SUBAPPLICATION Versuch_406 (* Versuch Array Summe *)
  (* Standard: 61499-2; Description: Copyright (c) 2023 Meisterschulen am Ostbahnhof This program and the accompanying materials are made available under the terms of the Eclipse Public License 2.0 which is available at https://www.eclipse.org/legal/epl-2.0/ SPDX-License-Identifier: EPL-2.0 *)
  (* Version 1.0, 2023-10-23, Franz Höpfinger, Meisterschulen am Ostbahnhof, initial API and implementation and/or initial documentation *)
  PACKAGE Versuche;
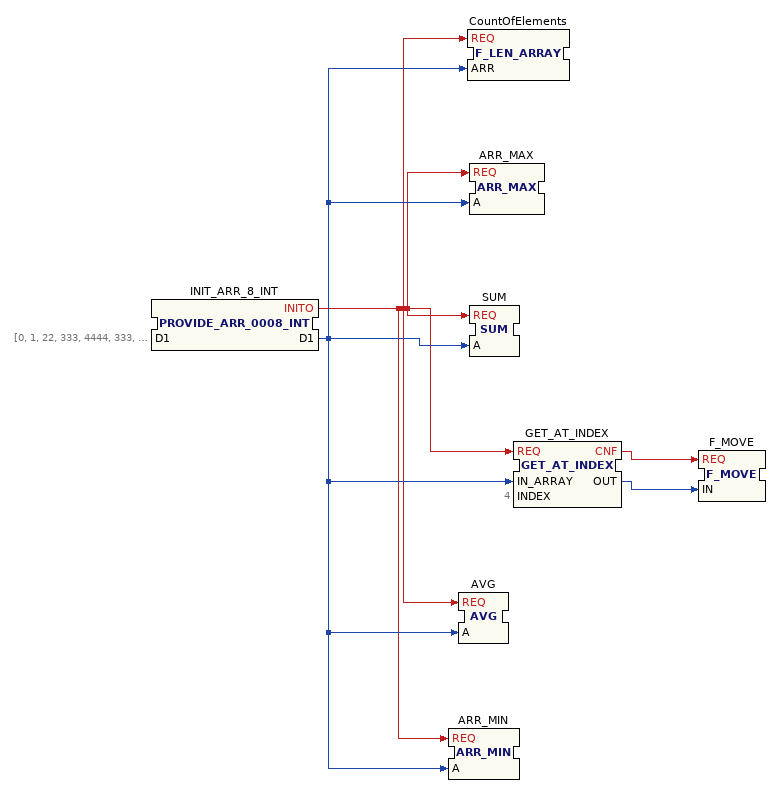
  FBS
    SUM : logiBUS::utils::dyn_arr::SUM;
    INIT_ARR_8_INT : eclipse4diac::convert::providers::PROVIDE_ARR_0008_INT(D1 := [0, 1, 22, 333, 4444, 333, 22, 1]);
    GET_AT_INDEX : eclipse4diac::convert::GET_AT_INDEX(INDEX := 4);
    F_MOVE : iec61131::selection::F_MOVE; {SET_ATTRIBUTE(DataType, INT)}
    ARR_MIN : logiBUS::utils::dyn_arr::ARR_MIN;
    ARR_MAX : logiBUS::utils::dyn_arr::ARR_MAX;
    AVG : logiBUS::utils::dyn_arr::AVG;
    CountOfElements : eclipse4diac::utils::arrays::F_LEN_ARRAY;
  END_FBS
  EVENT_CONNECTIONS
    GET_AT_INDEX.CNF TO F_MOVE.REQ;
    INIT_ARR_8_INT.INITO TO SUM.REQ;
    INIT_ARR_8_INT.INITO TO CountOfElements.REQ;
    INIT_ARR_8_INT.INITO TO ARR_MAX.REQ;
    INIT_ARR_8_INT.INITO TO GET_AT_INDEX.REQ;
    INIT_ARR_8_INT.INITO TO AVG.REQ;
    INIT_ARR_8_INT.INITO TO ARR_MIN.REQ;
  END_CONNECTIONS
  DATA_CONNECTIONS
    INIT_ARR_8_INT.D1 TO SUM.A;
    INIT_ARR_8_INT.D1 TO GET_AT_INDEX.IN_ARRAY;
    GET_AT_INDEX.OUT TO F_MOVE.IN;
    INIT_ARR_8_INT.D1 TO ARR_MIN.A;
    INIT_ARR_8_INT.D1 TO ARR_MAX.A;
    INIT_ARR_8_INT.D1 TO AVG.A;
    INIT_ARR_8_INT.D1 TO CountOfElements.ARR;
  END_CONNECTIONS
END_SUBAPPLICATION
